MOVL C09953 V=800.0 PL=0
MOVL C09954 V=800.0 PL=0
MOVL C09955 V=800.0 PL=0
MOVL C09956 V=800.0 PL=0
MOVL C09957 V=800.0 PL=0
MOVL C09958 V=800.0 PL=0
MOVL C09959 V=800.0 PL=0
MOVL C09960 V=800.0 PL=0
MOVL C09961 V=800.0 PL=0
MOVL C09962 V=800.0 PL=0
MOVL C09963 V=800.0 PL=0
MOVL C09964 V=800.0 PL=0
MOVL C09965 V=800.0 PL=0
MOVL C09966 V=800.0 PL=0
MOVL C09967 V=800.0 PL=0
MOVL C09968 V=800.0 PL=0
MOVL C09969 V=800.0 PL=0
MOVL C09970 V=800.0 PL=0
MOVL C09971 V=800.0 PL=0
MOVL C09972 V=800.0 PL=0
MOVL C09973 V=800.0 PL=0
MOVL C09974 V=800.0 PL=0
MOVL C09975 V=800.0 PL=0
MOVL C09976 V=800.0 PL=0
MOVL C09977 V=800.0 PL=0
MOVL C09978 V=800.0 PL=0
MOVL C09979 V=800.0 PL=0
MOVL C09980 V=800.0 PL=0
MOVL C09981 V=800.0 PL=0
MOVL C09982 V=800.0 PL=0
MOVL C09983 V=800.0 PL=0
MOVL C09984 V=800.0 PL=0
MOVL C09985 V=800.0 PL=0
MOVL C09986 V=800.0 PL=0
MOVL C09987 V=800.0 PL=0
MOVL C09988 V=800.0 PL=0
MOVL C09989 V=800.0 PL=0
MOVL C09990 V=800.0 PL=0
MOVL C09991 V=800.0 PL=0
MOVL C09992 V=800.0 PL=0
MOVL C09993 V=800.0 PL=0
MOVL C09994 V=800.0 PL=0
MOVL C09995 V=800.0 PL=0
MOVL C09996 V=800.0 PL=0
CALL JOB:A_ROOF_SIDE_0617_2_PAINT_24
END
